TYPE "PositioningMachine_DataPers"
VERSION : 0.1
// Block: PositioningMachine_DataPers
   STRUCT
      AxisEncoderSelection_OK : Bool;
      AxisParameters_OK : Bool;
      AxisReloadPostion_OK : Bool;
      ActualPosition : LReal;
   END_STRUCT;

END_TYPE
